// TIA Portal V19 export
FUNCTION_BLOCK "Positioning_DOL_Machine_FB"   // FB54, LAD
TITLE = OPEN LOOP POSITIONING AXIS WITH DRIVE S120 TEL.1
// stored: Access Published, MemoryReserve 100, SetENOAutomatically false
   VAR_INPUT
      AreaInterface : "AreaInterface";
      ZSI : "udt_ZoneSafetyInterface";
      DSI : "udt_DeviceSafetyInterface";
      Drive : "TAx_DriveInterface";
      DataIn : "Positioning_DOL_Machine_DataIn";
      CIn : "Positioning_DOL_Machine_CIn";
      Config : "Positioning_DOL_Machine_Config";
      HW_ID_TEL1 : HW_SUBMODULE;
   END_VAR
   VAR_OUTPUT
      MachineInterface { ExternalAccessible := 'False'; ExternalVisible := 'False'; ExternalWritable := 'False'} : "MachineInterface";
      DataOut : "Positioning_DOL_Machine_DataOut";
      COut : "Positioning_DOL_Machine_COut";
   END_VAR
   VAR_IN_OUT
      PosFeedback : "PosFbk_ITF";
      Par : "Positioning_DOL_Machine_Par";
      Pers_Data : "Positioning_DOL_Machine_Pers_Data";
      Warning : "Positioning_DOL_Machine_Wng";
      Alarm : "Positioning_DOL_Machine_Alr";
   END_VAR
   VAR
      InitDone : Bool := FALSE;
      Diag : Struct
         S120 : "TO_Diagnostic";
      END_STRUCT;
      HMI : Struct
         Sts { S7_SetPoint := 'True'} : "UDT_HMI-Sts_PosDOL-MchFB";
         B_Preset : Bool;
         B_Preset_UM2 : Bool;
         PresetPosition : LReal;
         TargetPosition : LReal;
      END_STRUCT;
      Sts : Struct
         Standstill : Bool;
         AlarmPresence : Bool;
         WarningPresence : Bool;
         Gen_Cnd : Bool;
         Minus_Cnd : Bool;
         Plus_Cnd : Bool;
         Pos_Cnd : Bool;
         Preset_Cnd : Bool;
         ActualPosition : LReal;
         Act_SysTime : DTL;
         Prv_SysTime : DTL;
      END_STRUCT;
      Ctrl : Struct
         StopDueDoorOpeningRequest : Bool;
         StopAborting : Bool;
         SafeMotionEnable : Bool;
         StopInPhase : Bool;
         StopProgrammed : Bool;
         Preset : Bool;
         Minus_Pos_Aut : Bool;
         Plus_Pos_Aut : Bool;
         Minus_Pos_Man : Bool;
         Plus_Pos_Man : Bool;
         Minus_Vel_Man : Bool;
         Plus_Vel_Man : Bool;
         MoveToPos_Aut : Bool;
         MoveToPos_Man : Bool;
         MoveToPos : Bool;
         Minus_Vel : Bool;
         Plus_Vel : Bool;
         Fan : Bool;
         Pos : LReal;
         Speed : LReal;
         SpeedPercentage : LReal;
      END_STRUCT;
      Ax : "OnOffAxis";
      S120 { S7_SetPoint := 'True'} : "SpeedMotor";
      Fan_M : "Motor";
      TON_NoPendingCmd : TON_TIME;
      TON_MinusCnd { S7_SetPoint := 'True'} : TON_TIME;
      TON_PlusCnd { S7_SetPoint := 'True'} : TON_TIME;
      TON_Fan_DelayOff : TON_TIME;
      TON_Brake_TimeOut : TON_TIME;
      S120_STW_TEL1 { ExternalAccessible := 'False'; ExternalVisible := 'False'; ExternalWritable := 'False'} : PD_TEL1_IN;
      S120_ZSW_TEL1 { ExternalAccessible := 'False'; ExternalVisible := 'False'; ExternalWritable := 'False'} : PD_TEL1_OUT;
      GETIO_STW_TEL1 { S7_SetPoint := 'True'} : GETIO;
      SETIO_ZSW_TEL1 { S7_SetPoint := 'True'} : SETIO;
      AUX : Struct
         PB_Minus : Bool;
         PB_Plus : Bool;
         PB_MoveToPos : Bool;
         B_Preset { ExternalAccessible := 'False'; ExternalVisible := 'False'; ExternalWritable := 'False'} : Bool;
         B_Preset_UM2 : Bool;
      END_STRUCT;
   END_VAR
   VAR_TEMP
      PE : Struct
         PB_Minus : Bool;
         PB_Plus : Bool;
         PB_MoveToPos : Bool;
         B_Preset : Bool;
         B_Preset_UM2 : Bool;
      END_STRUCT;
      RETVAL : Int;
      Req : Bool;
      REAL_value : Real;
   END_VAR
   VAR_TEMP   // added for the SCL form of the ladder/FBD networks
      _w1 : Bool;
      _w2 : Bool;
      _w3 : Bool;
      _w4 : Bool;
      _w5 : Bool;
   END_VAR
BEGIN

REGION Network 1 (SCL): Init
   IF NOT #InitDone THEN

       #InitDone := TRUE;

       #RETVAL := RD_SYS_T(#Sts.Act_SysTime);

       #Sts.Prv_SysTime := #Sts.Act_SysTime;

   END_IF;
END_REGION

REGION Network 2 (SCL): Reset
   IF #AreaInterface.RstAlarms THEN

       #Alarm.BrakeTimeOut := FALSE;
       #Alarm.S120_ComErr := FALSE;
       #Alarm.Ax_NotHomed := FALSE;

       #Warning.NotAutReady := FALSE;
       #Warning.MissingCnd_Minus := FALSE;
       #Warning.MissingCnd_Plus := FALSE;

   END_IF;
END_REGION

REGION Network 3 (SCL): Actual Position
   #Sts.ActualPosition := #PosFeedback.Sts.Position;
END_REGION

REGION Network 4: >
END_REGION

REGION Network 5: <<< MACHINE STOP >>>
END_REGION

REGION Network 6: Machine stop movements due door open request
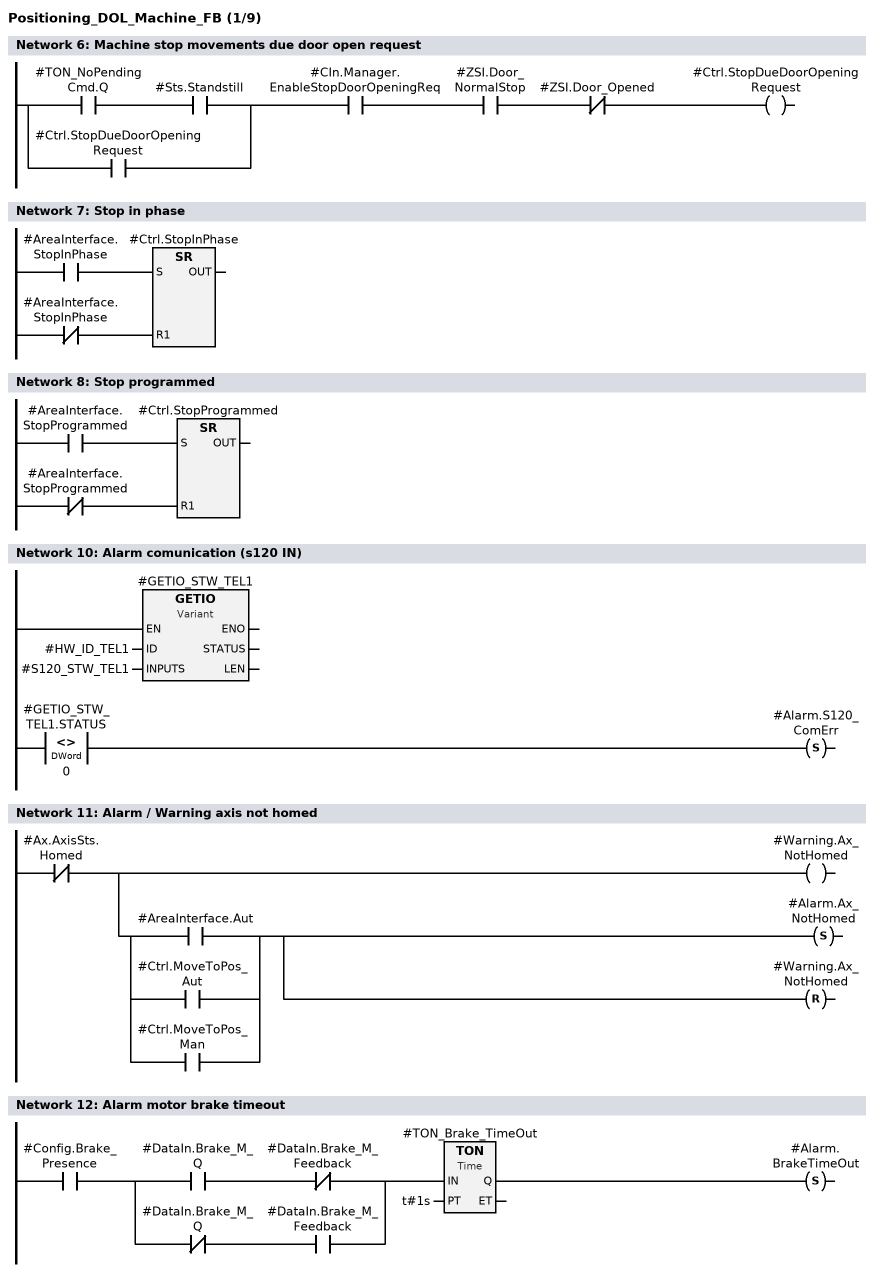
   RUNG wire#powerrail
      Contact( #TON_NoPendingCmd.Q )
      Contact( #Sts.Standstill )
      wire#w1
      Contact( #CIn.Manager.EnableStopDoorOpeningReq )
      Contact( #ZSI.Door_NormalStop )
      I_Contact( #ZSI.Door_Opened )
      Coil( #Ctrl.StopDueDoorOpeningRequest )
   END_RUNG
   RUNG wire#powerrail
      Contact( #Ctrl.StopDueDoorOpeningRequest )
   END_RUNG wire#w1
   // the same network as SCL:
   #Ctrl.StopDueDoorOpeningRequest := ((#TON_NoPendingCmd.Q AND #Sts.Standstill) OR #Ctrl.StopDueDoorOpeningRequest) AND #CIn.Manager.EnableStopDoorOpeningReq AND #ZSI.Door_NormalStop AND NOT #ZSI.Door_Opened;
END_REGION

REGION Network 7: Stop in phase
   RUNG wire#powerrail
      Contact( #AreaInterface.StopInPhase )
      S_SR(operand := #Ctrl.StopInPhase, r1 := wire#w1)
   END_RUNG
   RUNG wire#powerrail
      I_Contact( #AreaInterface.StopInPhase )
   END_RUNG wire#w1
   // the same network as SCL:
   IF #AreaInterface.StopInPhase THEN
       #Ctrl.StopInPhase := TRUE;   // SR flip-flop
   END_IF;
   IF NOT #AreaInterface.StopInPhase THEN #Ctrl.StopInPhase := FALSE; END_IF;
END_REGION

REGION Network 8: Stop programmed
   RUNG wire#powerrail
      Contact( #AreaInterface.StopProgrammed )
      S_SR(operand := #Ctrl.StopProgrammed, r1 := wire#w1)
   END_RUNG
   RUNG wire#powerrail
      I_Contact( #AreaInterface.StopProgrammed )
   END_RUNG wire#w1
   // the same network as SCL:
   IF #AreaInterface.StopProgrammed THEN
       #Ctrl.StopProgrammed := TRUE;   // SR flip-flop
   END_IF;
   IF NOT #AreaInterface.StopProgrammed THEN #Ctrl.StopProgrammed := FALSE; END_IF;
END_REGION

REGION Network 9: >
END_REGION

REGION Network 10: Alarm comunication (s120 IN)
   RUNG wire#powerrail
      { S7_Templates := "[ptr_type := Variant, id_type := HW_SUBMODULE]" } #GETIO_STW_TEL1.GETIO(ID := #HW_ID_TEL1, INPUTS := #S120_STW_TEL1, STATUS =>, LEN =>)
   END_RUNG
   RUNG wire#powerrail
      { S7_Templates := "SrcType := DWord" } NE_Contact(in1 := #GETIO_STW_TEL1.STATUS, in2 := 0)
      S_Coil( #Alarm.S120_ComErr )
   END_RUNG
   // the same network as SCL:
   #GETIO_STW_TEL1(ID := #HW_ID_TEL1, INPUTS := #S120_STW_TEL1);   // GETIO
   IF #GETIO_STW_TEL1.STATUS <> 0 THEN #Alarm.S120_ComErr := TRUE; END_IF;
END_REGION

REGION Network 11: Alarm / Warning axis not homed
   RUNG wire#powerrail
      I_Contact( #Ax.AxisSts.Homed )
      wire#w1
      Coil( #Warning.Ax_NotHomed )
   END_RUNG
   RUNG wire#w1
      Contact( #AreaInterface.Aut )
      wire#w2
      S_Coil( #Alarm.Ax_NotHomed )
   END_RUNG
   RUNG wire#w1
      Contact( #Ctrl.MoveToPos_Aut )
   END_RUNG wire#w2
   RUNG wire#w1
      Contact( #Ctrl.MoveToPos_Man )
   END_RUNG wire#w2
   RUNG wire#w2
      R_Coil( #Warning.Ax_NotHomed )
   END_RUNG
   // the same network as SCL:
   #Warning.Ax_NotHomed := NOT #Ax.AxisSts.Homed;
   IF NOT #Ax.AxisSts.Homed AND (#AreaInterface.Aut OR #Ctrl.MoveToPos_Aut OR #Ctrl.MoveToPos_Man) THEN
       #Alarm.Ax_NotHomed := TRUE;
       #Warning.Ax_NotHomed := FALSE;
   END_IF;
END_REGION

REGION Network 12: Alarm motor brake timeout
   RUNG wire#powerrail
      Contact( #Config.Brake_Presence )
      wire#w1
      Contact( #DataIn.Brake_M_Q )
      I_Contact( #DataIn.Brake_M_Feedback )
      wire#w2
      { S7_Templates := "time_type := Time" } #TON_Brake_TimeOut.TON(pt := t#1s, et =>)
      S_Coil( #Alarm.BrakeTimeOut )
   END_RUNG
   RUNG wire#w1
      I_Contact( #DataIn.Brake_M_Q )
      Contact( #DataIn.Brake_M_Feedback )
   END_RUNG wire#w2
   // the same network as SCL:
   #TON_Brake_TimeOut(IN := #Config.Brake_Presence AND ((#DataIn.Brake_M_Q AND NOT #DataIn.Brake_M_Feedback) OR (NOT #DataIn.Brake_M_Q AND #DataIn.Brake_M_Feedback)),   // TON
                      PT := t#1s);
   IF #TON_Brake_TimeOut.Q THEN #Alarm.BrakeTimeOut := TRUE; END_IF;
END_REGION

REGION Network 13: >
END_REGION

REGION Network 14: Buttons
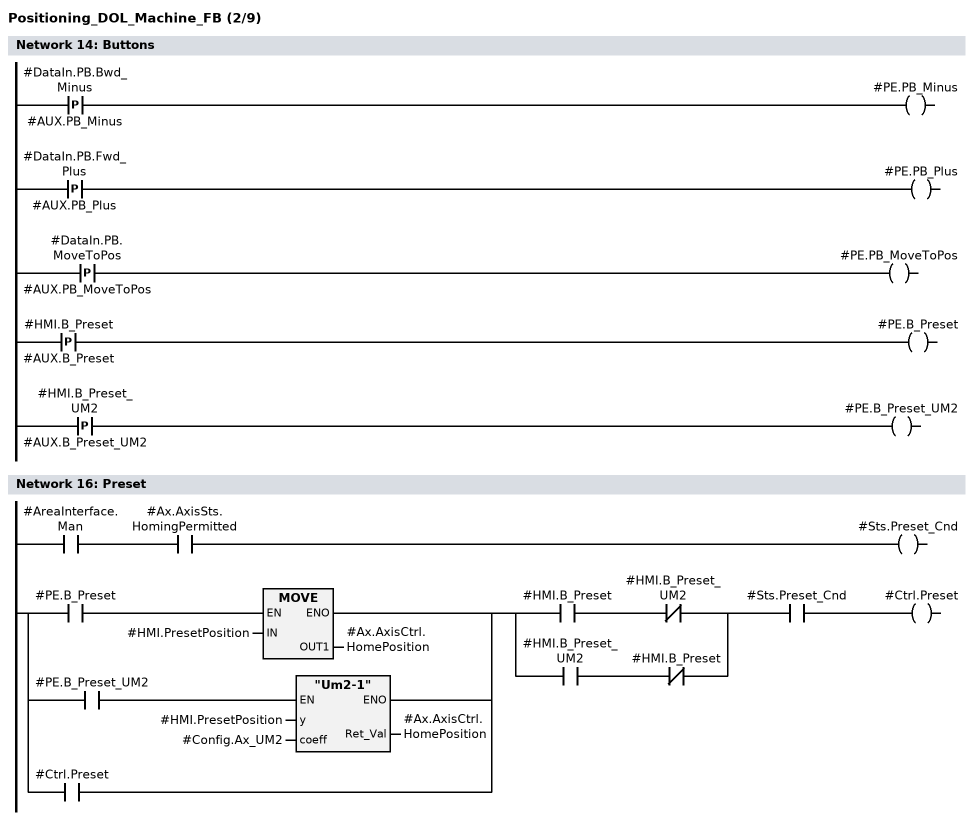
   RUNG wire#powerrail
      P_Contact(operand := #DataIn.PB.Bwd_Minus, bit := #AUX.PB_Minus)
      Coil( #PE.PB_Minus )
   END_RUNG
   RUNG wire#powerrail
      P_Contact(operand := #DataIn.PB.Fwd_Plus, bit := #AUX.PB_Plus)
      Coil( #PE.PB_Plus )
   END_RUNG
   RUNG wire#powerrail
      P_Contact(operand := #DataIn.PB.MoveToPos, bit := #AUX.PB_MoveToPos)
      Coil( #PE.PB_MoveToPos )
   END_RUNG
   RUNG wire#powerrail
      P_Contact(operand := #HMI.B_Preset, bit := #AUX.B_Preset)
      Coil( #PE.B_Preset )
   END_RUNG
   RUNG wire#powerrail
      P_Contact(operand := #HMI.B_Preset_UM2, bit := #AUX.B_Preset_UM2)
      Coil( #PE.B_Preset_UM2 )
   END_RUNG
   // the same network as SCL:
   #_w1 := #DataIn.PB.Bwd_Minus AND NOT #AUX.PB_Minus;   // rising edge of #DataIn.PB.Bwd_Minus
   #AUX.PB_Minus := #DataIn.PB.Bwd_Minus;
   #PE.PB_Minus := #_w1;
   #_w2 := #DataIn.PB.Fwd_Plus AND NOT #AUX.PB_Plus;   // rising edge of #DataIn.PB.Fwd_Plus
   #AUX.PB_Plus := #DataIn.PB.Fwd_Plus;
   #PE.PB_Plus := #_w2;
   #_w3 := #DataIn.PB.MoveToPos AND NOT #AUX.PB_MoveToPos;   // rising edge of #DataIn.PB.MoveToPos
   #AUX.PB_MoveToPos := #DataIn.PB.MoveToPos;
   #PE.PB_MoveToPos := #_w3;
   #_w4 := #HMI.B_Preset AND NOT #AUX.B_Preset;   // rising edge of #HMI.B_Preset
   #AUX.B_Preset := #HMI.B_Preset;
   #PE.B_Preset := #_w4;
   #_w5 := #HMI.B_Preset_UM2 AND NOT #AUX.B_Preset_UM2;   // rising edge of #HMI.B_Preset_UM2
   #AUX.B_Preset_UM2 := #HMI.B_Preset_UM2;
   #PE.B_Preset_UM2 := #_w5;
END_REGION

REGION Network 15: >
END_REGION

REGION Network 16: Preset
   RUNG wire#powerrail
      Contact( #AreaInterface.Man )
      Contact( #Ax.AxisSts.HomingPermitted )
      Coil( #Sts.Preset_Cnd )
   END_RUNG
   RUNG wire#powerrail
      Contact( #PE.B_Preset )
      Move(in := #HMI.PresetPosition, out1 => #Ax.AxisCtrl.HomePosition)
      wire#w1
      Contact( #HMI.B_Preset )
      I_Contact( #HMI.B_Preset_UM2 )
      wire#w2
      Contact( #Sts.Preset_Cnd )
      Coil( #Ctrl.Preset )
   END_RUNG
   RUNG wire#powerrail
      Contact( #PE.B_Preset_UM2 )
      "Um2-1"(y := #HMI.PresetPosition, coeff := #Config.Ax_UM2, Ret_Val => #Ax.AxisCtrl.HomePosition)
   END_RUNG wire#w1
   RUNG wire#powerrail
      Contact( #Ctrl.Preset )
   END_RUNG wire#w1
   RUNG wire#w1
      Contact( #HMI.B_Preset_UM2 )
      I_Contact( #HMI.B_Preset )
   END_RUNG wire#w2
   // the same network as SCL:
   #Sts.Preset_Cnd := #AreaInterface.Man AND #Ax.AxisSts.HomingPermitted;
   IF #PE.B_Preset THEN #Ax.AxisCtrl.HomePosition := #HMI.PresetPosition; END_IF;
   #Ax.AxisCtrl.HomePosition := "Um2-1"(EN := #PE.B_Preset_UM2,
                           y := #HMI.PresetPosition,
                           coeff := #Config.Ax_UM2,
                           ENO => #_w1);
   #Ctrl.Preset := (#PE.B_Preset OR #_w1 OR #Ctrl.Preset) AND ((#HMI.B_Preset AND NOT #HMI.B_Preset_UM2) OR (#HMI.B_Preset_UM2 AND NOT #HMI.B_Preset)) AND #Sts.Preset_Cnd;
END_REGION

REGION Network 17: Man
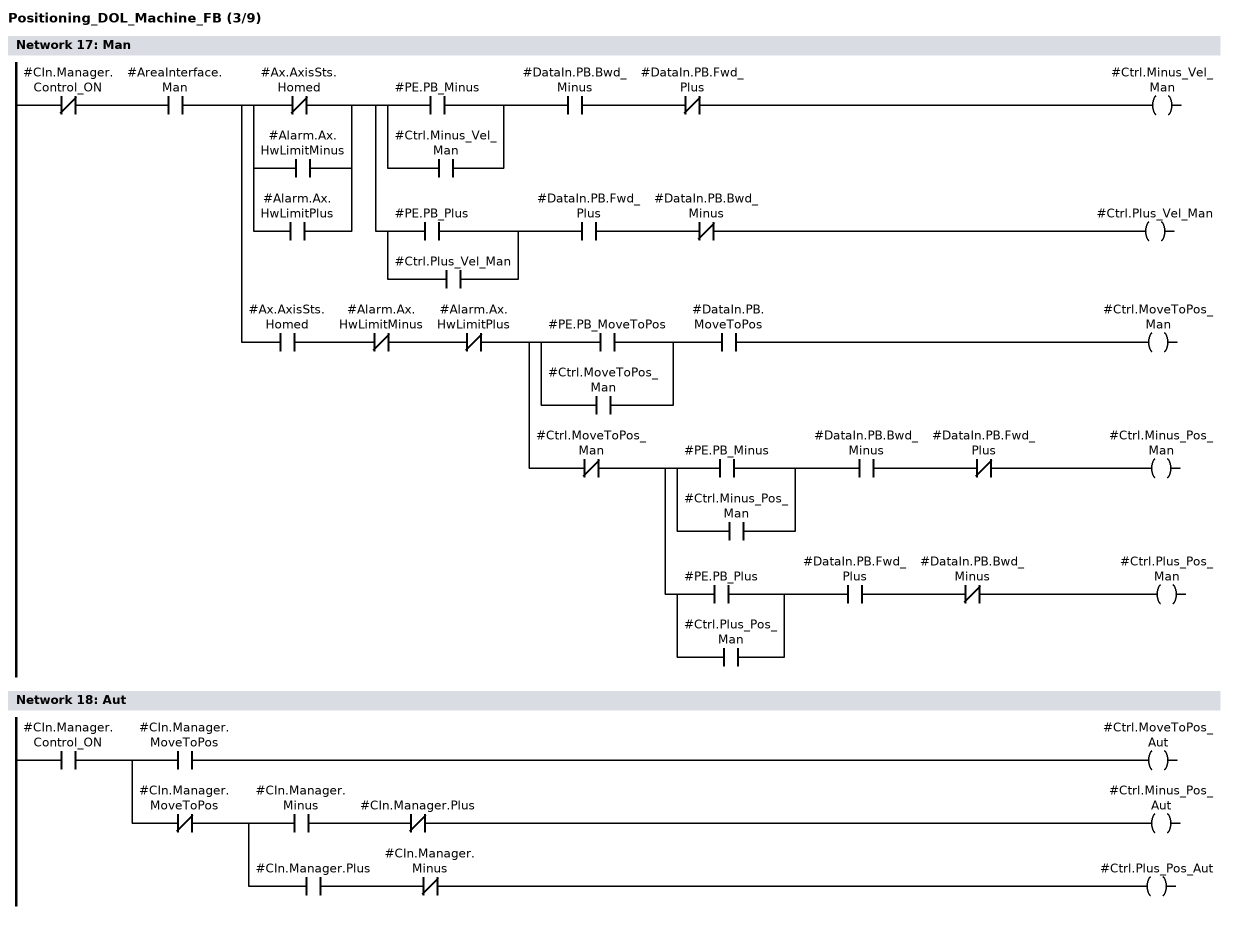
   RUNG wire#powerrail
      I_Contact( #CIn.Manager.Control_ON )
      Contact( #AreaInterface.Man )
      wire#w1
      I_Contact( #Ax.AxisSts.Homed )
      wire#w2
      Contact( #PE.PB_Minus )
      wire#w3
      Contact( #DataIn.PB.Bwd_Minus )
      I_Contact( #DataIn.PB.Fwd_Plus )
      Coil( #Ctrl.Minus_Vel_Man )
   END_RUNG
   RUNG wire#w1
      Contact( #Alarm.Ax.HwLimitMinus )
   END_RUNG wire#w2
   RUNG wire#w1
      Contact( #Alarm.Ax.HwLimitPlus )
   END_RUNG wire#w2
   RUNG wire#w2
      Contact( #Ctrl.Minus_Vel_Man )
   END_RUNG wire#w3
   RUNG wire#w2
      Contact( #PE.PB_Plus )
      wire#w4
      Contact( #DataIn.PB.Fwd_Plus )
      I_Contact( #DataIn.PB.Bwd_Minus )
      Coil( #Ctrl.Plus_Vel_Man )
   END_RUNG
   RUNG wire#w2
      Contact( #Ctrl.Plus_Vel_Man )
   END_RUNG wire#w4
   RUNG wire#w1
      Contact( #Ax.AxisSts.Homed )
      I_Contact( #Alarm.Ax.HwLimitMinus )
      I_Contact( #Alarm.Ax.HwLimitPlus )
      wire#w5
      Contact( #PE.PB_MoveToPos )
      wire#w6
      Contact( #DataIn.PB.MoveToPos )
      Coil( #Ctrl.MoveToPos_Man )
   END_RUNG
   RUNG wire#w5
      Contact( #Ctrl.MoveToPos_Man )
   END_RUNG wire#w6
   RUNG wire#w5
      I_Contact( #Ctrl.MoveToPos_Man )
      wire#w7
      Contact( #PE.PB_Minus )
      wire#w8
      Contact( #DataIn.PB.Bwd_Minus )
      I_Contact( #DataIn.PB.Fwd_Plus )
      Coil( #Ctrl.Minus_Pos_Man )
   END_RUNG
   RUNG wire#w7
      Contact( #Ctrl.Minus_Pos_Man )
   END_RUNG wire#w8
   RUNG wire#w7
      Contact( #PE.PB_Plus )
      wire#w9
      Contact( #DataIn.PB.Fwd_Plus )
      I_Contact( #DataIn.PB.Bwd_Minus )
      Coil( #Ctrl.Plus_Pos_Man )
   END_RUNG
   RUNG wire#w7
      Contact( #Ctrl.Plus_Pos_Man )
   END_RUNG wire#w9
   // the same network as SCL:
   #_w1 := NOT #CIn.Manager.Control_ON AND #AreaInterface.Man;
   #_w2 := #_w1 AND (NOT #Ax.AxisSts.Homed OR #Alarm.Ax.HwLimitMinus OR #Alarm.Ax.HwLimitPlus);
   #Ctrl.Minus_Vel_Man := #_w2 AND (#PE.PB_Minus OR #Ctrl.Minus_Vel_Man) AND #DataIn.PB.Bwd_Minus AND NOT #DataIn.PB.Fwd_Plus;
   #Ctrl.Plus_Vel_Man := #_w2 AND (#PE.PB_Plus OR #Ctrl.Plus_Vel_Man) AND #DataIn.PB.Fwd_Plus AND NOT #DataIn.PB.Bwd_Minus;
   #_w3 := #_w1 AND #Ax.AxisSts.Homed AND NOT #Alarm.Ax.HwLimitMinus AND NOT #Alarm.Ax.HwLimitPlus;
   #Ctrl.MoveToPos_Man := #_w3 AND (#PE.PB_MoveToPos OR #Ctrl.MoveToPos_Man) AND #DataIn.PB.MoveToPos;
   #_w4 := #_w3 AND NOT #Ctrl.MoveToPos_Man;
   #Ctrl.Minus_Pos_Man := #_w4 AND (#PE.PB_Minus OR #Ctrl.Minus_Pos_Man) AND #DataIn.PB.Bwd_Minus AND NOT #DataIn.PB.Fwd_Plus;
   #Ctrl.Plus_Pos_Man := #_w4 AND (#PE.PB_Plus OR #Ctrl.Plus_Pos_Man) AND #DataIn.PB.Fwd_Plus AND NOT #DataIn.PB.Bwd_Minus;
END_REGION

REGION Network 18: Aut
   RUNG wire#powerrail
      Contact( #CIn.Manager.Control_ON )
      wire#w1
      Contact( #CIn.Manager.MoveToPos )
      Coil( #Ctrl.MoveToPos_Aut )
   END_RUNG
   RUNG wire#w1
      I_Contact( #CIn.Manager.MoveToPos )
      wire#w2
      Contact( #CIn.Manager.Minus )
      I_Contact( #CIn.Manager.Plus )
      Coil( #Ctrl.Minus_Pos_Aut )
   END_RUNG
   RUNG wire#w2
      Contact( #CIn.Manager.Plus )
      I_Contact( #CIn.Manager.Minus )
      Coil( #Ctrl.Plus_Pos_Aut )
   END_RUNG
   // the same network as SCL:
   #Ctrl.MoveToPos_Aut := #CIn.Manager.Control_ON AND #CIn.Manager.MoveToPos;
   #_w1 := #CIn.Manager.Control_ON AND NOT #CIn.Manager.MoveToPos;
   #Ctrl.Minus_Pos_Aut := #_w1 AND #CIn.Manager.Minus AND NOT #CIn.Manager.Plus;
   #Ctrl.Plus_Pos_Aut := #_w1 AND #CIn.Manager.Plus AND NOT #CIn.Manager.Minus;
END_REGION

REGION Network 19: >
END_REGION

REGION Network 20 (SCL): Axis Limits
   #COut.MinPosition := #Par.Minus_Limit; //+ #Par.PosTolerance ; 

   #COut.MaxPosition := #Par.Plus_Limit; //- #Par.PosTolerance;


   IF #CIn.PositionLimits.EnableMin THEN
       #COut.MinPosition := MAX(IN1 := #COut.MinPosition, IN2 := #CIn.PositionLimits.PosMin);
   END_IF;

   IF #CIn.PositionLimits.EnableMax THEN
       #COut.MaxPosition := MIN(IN1 := #COut.MaxPosition, IN2 := #CIn.PositionLimits.PosMax);
   END_IF;
END_REGION

REGION Network 21 (SCL): Software Limit switches / External limits reached / exceed
   #COut.MinusLsSwReached := FALSE;
   #COut.PlusLsSwReached := FALSE;
   #COut.MinusLimitReached := FALSE;
   #COut.PlusLimitReached := FALSE;


   IF #Ax.AxisSts.Homed THEN

       #COut.MinusLsSwReached := #Warning.Ax.SwLimitMinus; //OR (ABS(#Sts.ActualPosition - #Par.Minus_Limit) <= #Par.PosTolerance);
       #COut.PlusLsSwReached := #Warning.Ax.SwLimitPlus; //OR (ABS(#Sts.ActualPosition - #Par.Plus_Limit) <= #Par.PosTolerance);


       IF NOT #COut.MinusLsSwReached AND #CIn.PositionLimits.EnableMin THEN

           #COut.MinusLimitReached := (#Sts.ActualPosition < #COut.MinPosition) OR (ABS(#Sts.ActualPosition - #COut.MinPosition) <= (#Par.PosTolerance/2));

       END_IF;



       IF NOT #COut.PlusLsSwReached  AND #CIn.PositionLimits.EnableMax THEN

           #COut.PlusLimitReached := (#Sts.ActualPosition > #COut.MaxPosition) OR (ABS(#Sts.ActualPosition - #COut.MaxPosition) <= (#Par.PosTolerance/2));

       END_IF;

   END_IF;
END_REGION

REGION Network 22 (SCL): Target position
   IF #CIn.Manager.Control_ON THEN


       #Ctrl.Pos := #CIn.Manager.Pos;

       IF #Ctrl.Minus_Pos_Aut THEN
           #Ctrl.Pos := #COut.MinPosition;

       ELSIF #Ctrl.Plus_Pos_Aut THEN
           #Ctrl.Pos := #COut.MaxPosition;
       END_IF;


       #HMI.TargetPosition := #Ctrl.Pos;

   ELSE


       #Ctrl.Pos := #HMI.TargetPosition;

       IF #Ctrl.Minus_Pos_Man THEN
           #Ctrl.Pos := #COut.MinPosition;
           #HMI.TargetPosition := #Ctrl.Pos;

       ELSIF #Ctrl.Plus_Pos_Man THEN
           #Ctrl.Pos := #COut.MaxPosition;
           #HMI.TargetPosition := #Ctrl.Pos;
       END_IF;

   END_IF;





   //---   



   // Dynamics limiting
   // 

   #Ctrl.Pos := LIMIT(IN := #Ctrl.Pos, MN := #COut.MinPosition, MX := #COut.MaxPosition);
END_REGION

REGION Network 23: >
END_REGION

REGION Network 24: Conditions
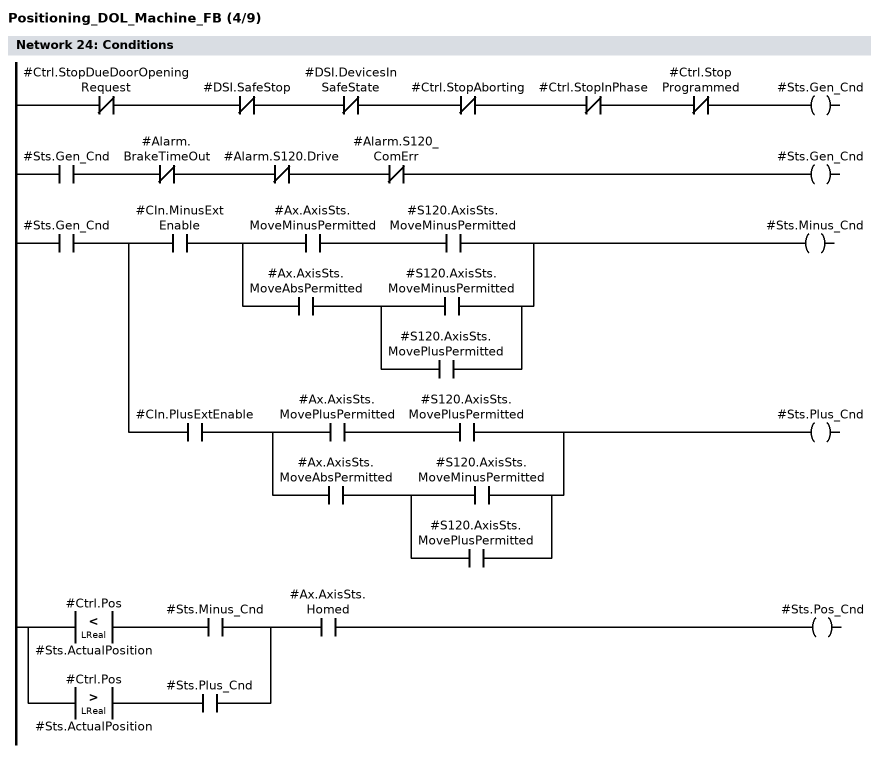
   RUNG wire#powerrail
      I_Contact( #Ctrl.StopDueDoorOpeningRequest )
      I_Contact( #DSI.SafeStop )
      I_Contact( #DSI.DevicesInSafeState )
      I_Contact( #Ctrl.StopAborting )
      I_Contact( #Ctrl.StopInPhase )
      I_Contact( #Ctrl.StopProgrammed )
      Coil( #Sts.Gen_Cnd )
   END_RUNG
   RUNG wire#powerrail
      Contact( #Sts.Gen_Cnd )
      I_Contact( #Alarm.BrakeTimeOut )
      I_Contact( #Alarm.S120.Drive )
      I_Contact( #Alarm.S120_ComErr )
      Coil( #Sts.Gen_Cnd )
   END_RUNG
   RUNG wire#powerrail
      Contact( #Sts.Gen_Cnd )
      wire#w1
      Contact( #CIn.MinusExtEnable )
      wire#w2
      Contact( #Ax.AxisSts.MoveMinusPermitted )
      Contact( #S120.AxisSts.MoveMinusPermitted )
      wire#w3
      Coil( #Sts.Minus_Cnd )
   END_RUNG
   RUNG wire#w2
      Contact( #Ax.AxisSts.MoveAbsPermitted )
      wire#w4
      Contact( #S120.AxisSts.MoveMinusPermitted )
   END_RUNG wire#w3
   RUNG wire#w4
      Contact( #S120.AxisSts.MovePlusPermitted )
   END_RUNG wire#w3
   RUNG wire#w1
      Contact( #CIn.PlusExtEnable )
      wire#w5
      Contact( #Ax.AxisSts.MovePlusPermitted )
      Contact( #S120.AxisSts.MovePlusPermitted )
      wire#w6
      Coil( #Sts.Plus_Cnd )
   END_RUNG
   RUNG wire#w5
      Contact( #Ax.AxisSts.MoveAbsPermitted )
      wire#w7
      Contact( #S120.AxisSts.MoveMinusPermitted )
   END_RUNG wire#w6
   RUNG wire#w7
      Contact( #S120.AxisSts.MovePlusPermitted )
   END_RUNG wire#w6
   RUNG wire#powerrail
      { S7_Templates := "SrcType := LReal" } LT_Contact(in1 := #Ctrl.Pos, in2 := #Sts.ActualPosition)
      Contact( #Sts.Minus_Cnd )
      wire#w8
      Contact( #Ax.AxisSts.Homed )
      Coil( #Sts.Pos_Cnd )
   END_RUNG
   RUNG wire#powerrail
      { S7_Templates := "SrcType := LReal" } GT_Contact(in1 := #Ctrl.Pos, in2 := #Sts.ActualPosition)
      Contact( #Sts.Plus_Cnd )
   END_RUNG wire#w8
   // the same network as SCL:
   #Sts.Gen_Cnd := NOT #Ctrl.StopDueDoorOpeningRequest AND NOT #DSI.SafeStop AND NOT #DSI.DevicesInSafeState AND NOT #Ctrl.StopAborting AND NOT #Ctrl.StopInPhase AND NOT #Ctrl.StopProgrammed;
   #Sts.Gen_Cnd := #Sts.Gen_Cnd AND NOT #Alarm.BrakeTimeOut AND NOT #Alarm.S120.Drive AND NOT #Alarm.S120_ComErr;
   #Sts.Minus_Cnd := #Sts.Gen_Cnd AND #CIn.MinusExtEnable AND ((#Ax.AxisSts.MoveMinusPermitted AND #S120.AxisSts.MoveMinusPermitted) OR (#Ax.AxisSts.MoveAbsPermitted AND (#S120.AxisSts.MoveMinusPermitted OR #S120.AxisSts.MovePlusPermitted)));
   #Sts.Plus_Cnd := #Sts.Gen_Cnd AND #CIn.PlusExtEnable AND ((#Ax.AxisSts.MovePlusPermitted AND #S120.AxisSts.MovePlusPermitted) OR (#Ax.AxisSts.MoveAbsPermitted AND (#S120.AxisSts.MoveMinusPermitted OR #S120.AxisSts.MovePlusPermitted)));
   #Sts.Pos_Cnd := (((#Ctrl.Pos < #Sts.ActualPosition) AND #Sts.Minus_Cnd) OR ((#Ctrl.Pos > #Sts.ActualPosition) AND #Sts.Plus_Cnd)) AND #Ax.AxisSts.Homed;
END_REGION

REGION Network 25: >
END_REGION

REGION Network 26: <<< ON/OFF AXIS >>>
END_REGION

REGION Network 27: On/Off Axis - Controls
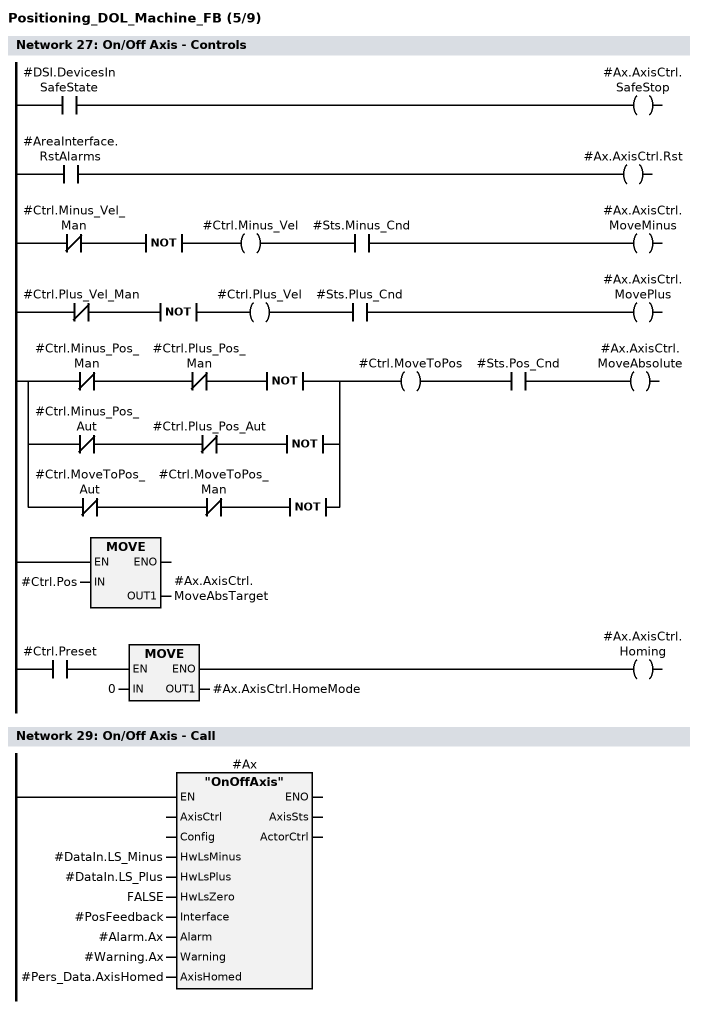
   RUNG wire#powerrail
      Contact( #DSI.DevicesInSafeState )
      Coil( #Ax.AxisCtrl.SafeStop )
   END_RUNG
   RUNG wire#powerrail
      Contact( #AreaInterface.RstAlarms )
      Coil( #Ax.AxisCtrl.Rst )
   END_RUNG
   RUNG wire#powerrail
      I_Contact( #Ctrl.Minus_Vel_Man )
      Not()
      Coil( #Ctrl.Minus_Vel )
      Contact( #Sts.Minus_Cnd )
      Coil( #Ax.AxisCtrl.MoveMinus )
   END_RUNG
   RUNG wire#powerrail
      I_Contact( #Ctrl.Plus_Vel_Man )
      Not()
      Coil( #Ctrl.Plus_Vel )
      Contact( #Sts.Plus_Cnd )
      Coil( #Ax.AxisCtrl.MovePlus )
   END_RUNG
   RUNG wire#powerrail
      I_Contact( #Ctrl.Minus_Pos_Man )
      I_Contact( #Ctrl.Plus_Pos_Man )
      Not()
      wire#w1
      Coil( #Ctrl.MoveToPos )
      Contact( #Sts.Pos_Cnd )
      Coil( #Ax.AxisCtrl.MoveAbsolute )
   END_RUNG
   RUNG wire#powerrail
      I_Contact( #Ctrl.Minus_Pos_Aut )
      I_Contact( #Ctrl.Plus_Pos_Aut )
      Not()
   END_RUNG wire#w1
   RUNG wire#powerrail
      I_Contact( #Ctrl.MoveToPos_Aut )
      I_Contact( #Ctrl.MoveToPos_Man )
      Not()
   END_RUNG wire#w1
   RUNG wire#powerrail
      Move(in := #Ctrl.Pos, out1 => #Ax.AxisCtrl.MoveAbsTarget)
   END_RUNG
   RUNG wire#powerrail
      Contact( #Ctrl.Preset )
      Move(in := 0, out1 => #Ax.AxisCtrl.HomeMode)
      Coil( #Ax.AxisCtrl.Homing )
   END_RUNG
   // the same network as SCL:
   #Ax.AxisCtrl.SafeStop := #DSI.DevicesInSafeState;
   #Ax.AxisCtrl.Rst := #AreaInterface.RstAlarms;
   #Ctrl.Minus_Vel := NOT (NOT #Ctrl.Minus_Vel_Man);
   #Ax.AxisCtrl.MoveMinus := NOT (NOT #Ctrl.Minus_Vel_Man) AND #Sts.Minus_Cnd;
   #Ctrl.Plus_Vel := NOT (NOT #Ctrl.Plus_Vel_Man);
   #Ax.AxisCtrl.MovePlus := NOT (NOT #Ctrl.Plus_Vel_Man) AND #Sts.Plus_Cnd;
   #Ctrl.MoveToPos := NOT (NOT #Ctrl.Minus_Pos_Man AND NOT #Ctrl.Plus_Pos_Man) OR NOT (NOT #Ctrl.Minus_Pos_Aut AND NOT #Ctrl.Plus_Pos_Aut) OR NOT (NOT #Ctrl.MoveToPos_Aut AND NOT #Ctrl.MoveToPos_Man);
   #Ax.AxisCtrl.MoveAbsolute := #Ctrl.MoveToPos AND #Sts.Pos_Cnd;
   #Ax.AxisCtrl.MoveAbsTarget := #Ctrl.Pos;
   IF #Ctrl.Preset THEN #Ax.AxisCtrl.HomeMode := 0; END_IF;
   #Ax.AxisCtrl.Homing := #Ctrl.Preset;
END_REGION

REGION Network 28 (SCL): On/Off Axis - Configuration
   #Ax.Config := #Config.Ax;

   #Ax.Config.limitMinus := #Par.Minus_Limit;
   #Ax.Config.limitPlus := #Par.Plus_Limit;

   #Ax.Config.ToleranceWindow := #Par.PosTolerance;
   #Ax.Config.PreCutOff := #Par.PreCutOff;
   #Ax.Config.PreEndMedSpeed := #Par.PreEndMedSpeed;
   #Ax.Config.PreEndLowSpeed := #Par.PreEndLowSpeed;


   #Ax.Config.StandStillDelay := DINT_TO_TIME(LREAL_TO_DINT(#Config.S120.DecTime + 0.1));



   IF #Config.CyclicOBTime_ms <= 0.0 THEN

       #Sts.Prv_SysTime := #Sts.Act_SysTime;

       #RETVAL := RD_SYS_T(#Sts.Act_SysTime);

       #Ax.Config.RecallTime := UDINT_TO_LREAL(TIME_TO_UDINT(T_DIFF(IN1 := #Sts.Act_SysTime, IN2 := #Sts.Prv_SysTime)));
       IF #Ax.Config.RecallTime <= 1 THEN
           #Ax.Config.RecallTime := 1;
       END_IF;
   ELSE

       #Ax.Config.RecallTime := #Config.CyclicOBTime_ms;

   END_IF;
END_REGION

REGION Network 29: On/Off Axis - Call
   RUNG wire#powerrail
      #Ax(AxisCtrl :=, Config :=, HwLsMinus := #DataIn.LS_Minus, HwLsPlus := #DataIn.LS_Plus, HwLsZero := FALSE, Interface := #PosFeedback, Alarm := #Alarm.Ax, Warning := #Warning.Ax, AxisHomed := #Pers_Data.AxisHomed, AxisSts =>, ActorCtrl =>)
   END_RUNG
   // the same network as SCL:
   #Ax(HwLsMinus := #DataIn.LS_Minus,   // "OnOffAxis"
       HwLsPlus := #DataIn.LS_Plus,
       HwLsZero := FALSE,
       Interface := #PosFeedback,
       Alarm := #Alarm.Ax,
       Warning := #Warning.Ax,
       AxisHomed := #Pers_Data.AxisHomed);
END_REGION

REGION Network 30 (SCL): On/Off Axis -Reset Wanrning

   #Warning.Ax.SwLimitMinus := (ABS(#Sts.ActualPosition - #Par.Minus_Limit) <= (#Par.PosTolerance / 2));
   #Warning.Ax.SwLimitPlus := (ABS(#Sts.ActualPosition - #Par.Plus_Limit) <= (#Par.PosTolerance / 2));
END_REGION

REGION Network 31 (SCL): S120 - Velocity & Dynamics
   #Ctrl.SpeedPercentage := #Par.Man_Speed;

   IF #CIn.Manager.Control_ON THEN
       #Ctrl.SpeedPercentage := #CIn.Manager.Speed;
   END_IF;

   #Ctrl.SpeedPercentage := MIN(IN1 := #Ctrl.SpeedPercentage, IN2 := 100.0);
   #Ctrl.SpeedPercentage := MAX(IN1 := #Ctrl.SpeedPercentage, IN2 := 0.0);


   #Ctrl.Speed := 0.0;


   IF #Ax.ActorCtrl.CmdLowSpeed THEN

       #Ctrl.Speed := (#Par.LowSpeed / 100.0) * #Config.S120.SpeedMotor.ReferenceVelocity;


       IF NOT #Ax.AxisCtrl.MoveAbsolute THEN

           #Ctrl.Speed := #Ctrl.Speed * #Ctrl.SpeedPercentage / 100.0;
       END_IF;


   ELSIF #Ax.ActorCtrl.CmdMediumSpeed THEN

       #Ctrl.Speed := (#Par.MedSpeed / 100.0) * #Config.S120.SpeedMotor.ReferenceVelocity;

       #Ctrl.Speed := #Ctrl.Speed * #Ctrl.SpeedPercentage / 100.0;


   ELSIF #Ax.ActorCtrl.CmdHighSpeed THEN

       #Ctrl.Speed := (#Par.HighSpeed / 100.0) * #Config.S120.SpeedMotor.ReferenceVelocity;

       #Ctrl.Speed := #Ctrl.Speed * #Ctrl.SpeedPercentage / 100.0;
   END_IF;



   // Brake not open... Velocity  = 0.0
   // 
   IF #Config.Brake_Presence AND NOT #DataIn.Brake_M_Feedback THEN
       #Ctrl.Speed := 0.0;
   END_IF;



   #S120.AxisCtrl.Velocity := MIN(IN1 := #Ctrl.Speed , IN2 := #Config.S120.SpeedMotor.ReferenceVelocity);

   #S120.AxisCtrl.Acceleration := #Config.S120.SpeedMotor.ReferenceVelocity / 60.0 / #Config.S120.AccTime;
   #S120.AxisCtrl.Deceleration := #Config.S120.SpeedMotor.ReferenceVelocity / 60.0 / #Config.S120.DecTime;
END_REGION

REGION Network 32: S120 - Control
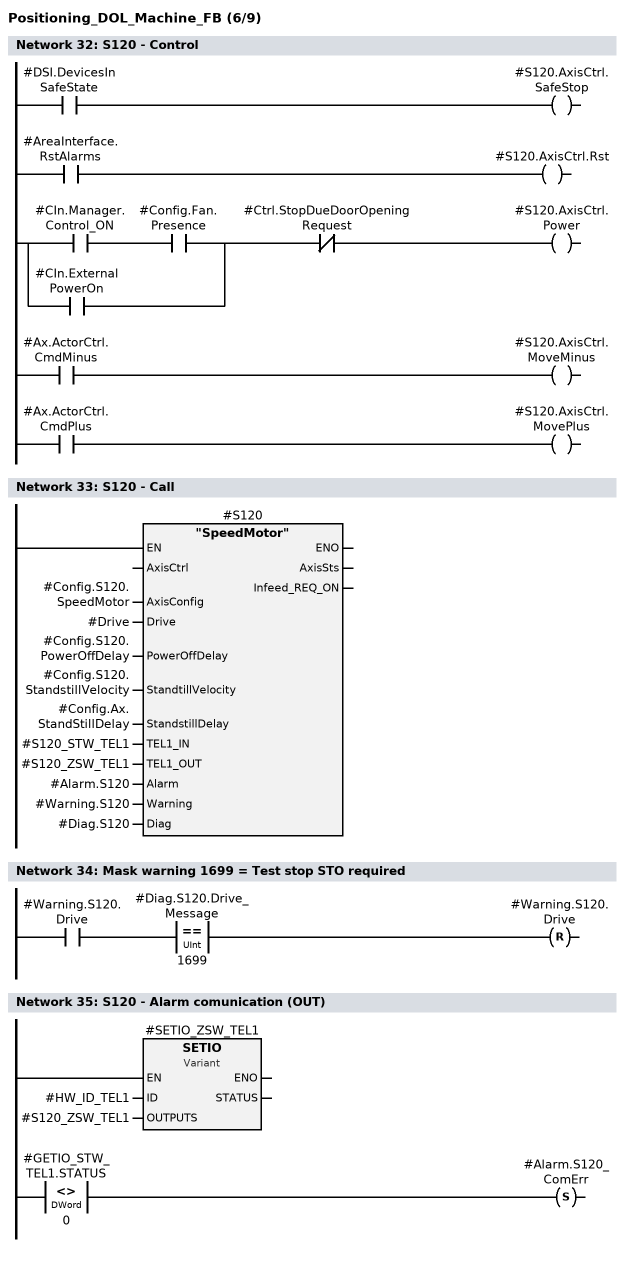
   RUNG wire#powerrail
      Contact( #DSI.DevicesInSafeState )
      Coil( #S120.AxisCtrl.SafeStop )
   END_RUNG
   RUNG wire#powerrail
      Contact( #AreaInterface.RstAlarms )
      Coil( #S120.AxisCtrl.Rst )
   END_RUNG
   RUNG wire#powerrail
      Contact( #CIn.Manager.Control_ON )
      Contact( #Config.Fan.Presence )
      wire#w1
      I_Contact( #Ctrl.StopDueDoorOpeningRequest )
      Coil( #S120.AxisCtrl.Power )
   END_RUNG
   RUNG wire#powerrail
      Contact( #CIn.ExternalPowerOn )
   END_RUNG wire#w1
   RUNG wire#powerrail
      Contact( #Ax.ActorCtrl.CmdMinus )
      Coil( #S120.AxisCtrl.MoveMinus )
   END_RUNG
   RUNG wire#powerrail
      Contact( #Ax.ActorCtrl.CmdPlus )
      Coil( #S120.AxisCtrl.MovePlus )
   END_RUNG
   // the same network as SCL:
   #S120.AxisCtrl.SafeStop := #DSI.DevicesInSafeState;
   #S120.AxisCtrl.Rst := #AreaInterface.RstAlarms;
   #S120.AxisCtrl.Power := ((#CIn.Manager.Control_ON AND #Config.Fan.Presence) OR #CIn.ExternalPowerOn) AND NOT #Ctrl.StopDueDoorOpeningRequest;
   #S120.AxisCtrl.MoveMinus := #Ax.ActorCtrl.CmdMinus;
   #S120.AxisCtrl.MovePlus := #Ax.ActorCtrl.CmdPlus;
END_REGION

REGION Network 33: S120 - Call
   RUNG wire#powerrail
      #S120(AxisCtrl :=, AxisConfig := #Config.S120.SpeedMotor, Drive := #Drive, PowerOffDelay := #Config.S120.PowerOffDelay, StandtillVelocity := #Config.S120.StandstillVelocity, StandstillDelay := #Config.Ax.StandStillDelay, TEL1_IN := #S120_STW_TEL1, TEL1_OUT := #S120_ZSW_TEL1, Alarm := #Alarm.S120, Warning := #Warning.S120, Diag := #Diag.S120, AxisSts =>, Infeed_REQ_ON =>)
   END_RUNG
   // the same network as SCL:
   #S120(AxisConfig := #Config.S120.SpeedMotor,   // "SpeedMotor"
         Drive := #Drive,
         PowerOffDelay := #Config.S120.PowerOffDelay,
         StandtillVelocity := #Config.S120.StandstillVelocity,
         StandstillDelay := #Config.Ax.StandStillDelay,
         TEL1_IN := #S120_STW_TEL1,
         TEL1_OUT := #S120_ZSW_TEL1,
         Alarm := #Alarm.S120,
         Warning := #Warning.S120,
         Diag := #Diag.S120);
END_REGION

REGION Network 34: Mask warning 1699 = Test stop STO required
   RUNG wire#powerrail
      Contact( #Warning.S120.Drive )
      { S7_Templates := "SrcType := UInt" } EQ_Contact(in1 := #Diag.S120.Drive_Message, in2 := 1699)
      R_Coil( #Warning.S120.Drive )
   END_RUNG
   // the same network as SCL:
   IF #Warning.S120.Drive AND (#Diag.S120.Drive_Message = 1699) THEN #Warning.S120.Drive := FALSE; END_IF;
END_REGION

REGION Network 35: S120 - Alarm comunication (OUT)
   RUNG wire#powerrail
      { S7_Templates := "[card := 0, ptr_type := Variant, id_type := HW_SUBMODULE]" } #SETIO_ZSW_TEL1.SETIO(ID := #HW_ID_TEL1, OUTPUTS := #S120_ZSW_TEL1, STATUS =>)
   END_RUNG
   RUNG wire#powerrail
      { S7_Templates := "SrcType := DWord" } NE_Contact(in1 := #GETIO_STW_TEL1.STATUS, in2 := 0)
      S_Coil( #Alarm.S120_ComErr )
   END_RUNG
   // the same network as SCL:
   #SETIO_ZSW_TEL1(ID := #HW_ID_TEL1, OUTPUTS := #S120_ZSW_TEL1);   // SETIO
   IF #GETIO_STW_TEL1.STATUS <> 0 THEN #Alarm.S120_ComErr := TRUE; END_IF;
END_REGION

REGION Network 36: <<< MOTOR FAN >>>
END_REGION

REGION Network 37: Run
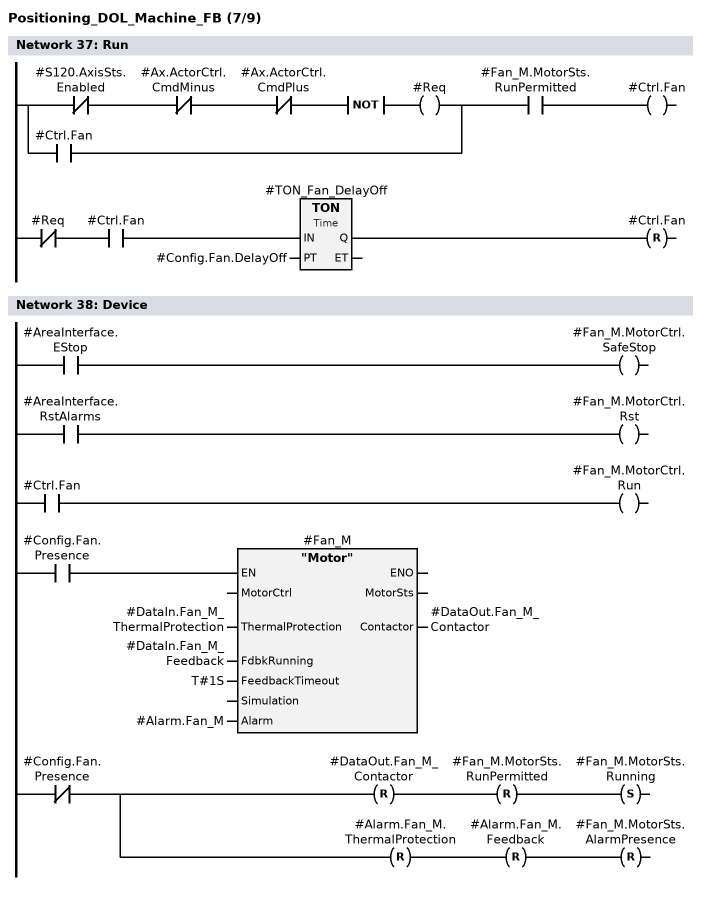
   RUNG wire#powerrail
      I_Contact( #S120.AxisSts.Enabled )
      I_Contact( #Ax.ActorCtrl.CmdMinus )
      I_Contact( #Ax.ActorCtrl.CmdPlus )
      Not()
      Coil( #Req )
      wire#w1
      Contact( #Fan_M.MotorSts.RunPermitted )
      Coil( #Ctrl.Fan )
   END_RUNG
   RUNG wire#powerrail
      Contact( #Ctrl.Fan )
   END_RUNG wire#w1
   RUNG wire#powerrail
      I_Contact( #Req )
      Contact( #Ctrl.Fan )
      { S7_Templates := "time_type := Time" } #TON_Fan_DelayOff.TON(pt := #Config.Fan.DelayOff, et =>)
      R_Coil( #Ctrl.Fan )
   END_RUNG
   // the same network as SCL:
   #Req := NOT (NOT #S120.AxisSts.Enabled AND NOT #Ax.ActorCtrl.CmdMinus AND NOT #Ax.ActorCtrl.CmdPlus);
   #Ctrl.Fan := (#Req OR #Ctrl.Fan) AND #Fan_M.MotorSts.RunPermitted;
   #TON_Fan_DelayOff(IN := NOT #Req AND #Ctrl.Fan, PT := #Config.Fan.DelayOff);   // TON
   IF #TON_Fan_DelayOff.Q THEN #Ctrl.Fan := FALSE; END_IF;
END_REGION

REGION Network 38: Device
   RUNG wire#powerrail
      Contact( #AreaInterface.EStop )
      Coil( #Fan_M.MotorCtrl.SafeStop )
   END_RUNG
   RUNG wire#powerrail
      Contact( #AreaInterface.RstAlarms )
      Coil( #Fan_M.MotorCtrl.Rst )
   END_RUNG
   RUNG wire#powerrail
      Contact( #Ctrl.Fan )
      Coil( #Fan_M.MotorCtrl.Run )
   END_RUNG
   RUNG wire#powerrail
      Contact( #Config.Fan.Presence )
      #Fan_M(MotorCtrl :=, ThermalProtection := #DataIn.Fan_M_ThermalProtection, FdbkRunning := #DataIn.Fan_M_Feedback, FeedbackTimeout := T#1S, Simulation :=, Alarm := #Alarm.Fan_M, MotorSts =>, Contactor => #DataOut.Fan_M_Contactor)
   END_RUNG
   RUNG wire#powerrail
      I_Contact( #Config.Fan.Presence )
      wire#w1
      R_Coil( #DataOut.Fan_M_Contactor )
      R_Coil( #Fan_M.MotorSts.RunPermitted )
      S_Coil( #Fan_M.MotorSts.Running )
   END_RUNG
   RUNG wire#w1
      R_Coil( #Alarm.Fan_M.ThermalProtection )
      R_Coil( #Alarm.Fan_M.Feedback )
      R_Coil( #Fan_M.MotorSts.AlarmPresence )
   END_RUNG
   // the same network as SCL:
   #Fan_M.MotorCtrl.SafeStop := #AreaInterface.EStop;
   #Fan_M.MotorCtrl.Rst := #AreaInterface.RstAlarms;
   #Fan_M.MotorCtrl.Run := #Ctrl.Fan;
   IF #Config.Fan.Presence THEN
       #Fan_M(ThermalProtection := #DataIn.Fan_M_ThermalProtection,   // "Motor"
              FdbkRunning := #DataIn.Fan_M_Feedback,
              FeedbackTimeout := T#1S,
              Alarm := #Alarm.Fan_M,
              Contactor => #DataOut.Fan_M_Contactor);
   END_IF;
   IF NOT #Config.Fan.Presence THEN
       #DataOut.Fan_M_Contactor := FALSE;
       #Fan_M.MotorSts.RunPermitted := FALSE;
       #Fan_M.MotorSts.Running := TRUE;
       #Alarm.Fan_M.ThermalProtection := FALSE;
       #Alarm.Fan_M.Feedback := FALSE;
       #Fan_M.MotorSts.AlarmPresence := FALSE;
   END_IF;
END_REGION

REGION Network 39: >
END_REGION

REGION Network 40: >
END_REGION

REGION Network 41: Coordination Out
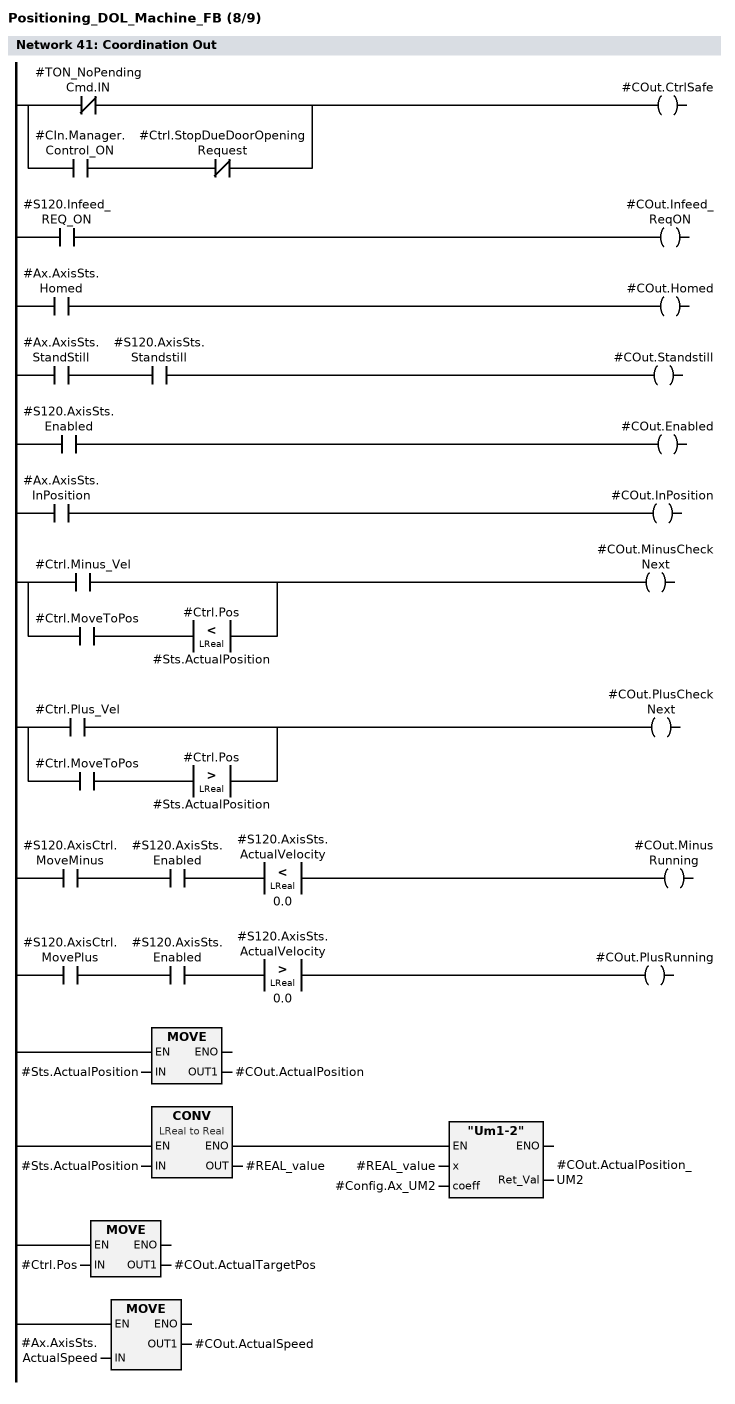
   RUNG wire#powerrail
      I_Contact( #TON_NoPendingCmd.IN )
      wire#w1
      Coil( #COut.CtrlSafe )
   END_RUNG
   RUNG wire#powerrail
      Contact( #CIn.Manager.Control_ON )
      I_Contact( #Ctrl.StopDueDoorOpeningRequest )
   END_RUNG wire#w1
   RUNG wire#powerrail
      Contact( #S120.Infeed_REQ_ON )
      Coil( #COut.Infeed_ReqON )
   END_RUNG
   RUNG wire#powerrail
      Contact( #Ax.AxisSts.Homed )
      Coil( #COut.Homed )
   END_RUNG
   RUNG wire#powerrail
      Contact( #Ax.AxisSts.StandStill )
      Contact( #S120.AxisSts.Standstill )
      Coil( #COut.Standstill )
   END_RUNG
   RUNG wire#powerrail
      Contact( #S120.AxisSts.Enabled )
      Coil( #COut.Enabled )
   END_RUNG
   RUNG wire#powerrail
      Contact( #Ax.AxisSts.InPosition )
      Coil( #COut.InPosition )
   END_RUNG
   RUNG wire#powerrail
      Contact( #Ctrl.Minus_Vel )
      wire#w2
      Coil( #COut.MinusCheckNext )
   END_RUNG
   RUNG wire#powerrail
      Contact( #Ctrl.MoveToPos )
      { S7_Templates := "SrcType := LReal" } LT_Contact(in1 := #Ctrl.Pos, in2 := #Sts.ActualPosition)
   END_RUNG wire#w2
   RUNG wire#powerrail
      Contact( #Ctrl.Plus_Vel )
      wire#w3
      Coil( #COut.PlusCheckNext )
   END_RUNG
   RUNG wire#powerrail
      Contact( #Ctrl.MoveToPos )
      { S7_Templates := "SrcType := LReal" } GT_Contact(in1 := #Ctrl.Pos, in2 := #Sts.ActualPosition)
   END_RUNG wire#w3
   RUNG wire#powerrail
      Contact( #S120.AxisCtrl.MoveMinus )
      Contact( #S120.AxisSts.Enabled )
      { S7_Templates := "SrcType := LReal" } LT_Contact(in1 := #S120.AxisSts.ActualVelocity, in2 := 0.0)
      Coil( #COut.MinusRunning )
   END_RUNG
   RUNG wire#powerrail
      Contact( #S120.AxisCtrl.MovePlus )
      Contact( #S120.AxisSts.Enabled )
      { S7_Templates := "SrcType := LReal" } GT_Contact(in1 := #S120.AxisSts.ActualVelocity, in2 := 0.0)
      Coil( #COut.PlusRunning )
   END_RUNG
   RUNG wire#powerrail
      Move(in := #Sts.ActualPosition, out1 => #COut.ActualPosition)
   END_RUNG
   RUNG wire#powerrail
      { S7_Templates := "[SrcType := LReal, DestType := Real]" } Convert(in := #Sts.ActualPosition, out => #REAL_value)
      "Um1-2"(x := #REAL_value, coeff := #Config.Ax_UM2, Ret_Val => #COut.ActualPosition_UM2)
   END_RUNG
   RUNG wire#powerrail
      Move(in := #Ctrl.Pos, out1 => #COut.ActualTargetPos)
   END_RUNG
   RUNG wire#powerrail
      Move(in := #Ax.AxisSts.ActualSpeed, out1 => #COut.ActualSpeed)
   END_RUNG
   // the same network as SCL:
   #COut.CtrlSafe := NOT #TON_NoPendingCmd.IN OR (#CIn.Manager.Control_ON AND NOT #Ctrl.StopDueDoorOpeningRequest);
   #COut.Infeed_ReqON := #S120.Infeed_REQ_ON;
   #COut.Homed := #Ax.AxisSts.Homed;
   #COut.Standstill := #Ax.AxisSts.StandStill AND #S120.AxisSts.Standstill;
   #COut.Enabled := #S120.AxisSts.Enabled;
   #COut.InPosition := #Ax.AxisSts.InPosition;
   #COut.MinusCheckNext := #Ctrl.Minus_Vel OR (#Ctrl.MoveToPos AND (#Ctrl.Pos < #Sts.ActualPosition));
   #COut.PlusCheckNext := #Ctrl.Plus_Vel OR (#Ctrl.MoveToPos AND (#Ctrl.Pos > #Sts.ActualPosition));
   #COut.MinusRunning := #S120.AxisCtrl.MoveMinus AND #S120.AxisSts.Enabled AND (#S120.AxisSts.ActualVelocity < 0.0);
   #COut.PlusRunning := #S120.AxisCtrl.MovePlus AND #S120.AxisSts.Enabled AND (#S120.AxisSts.ActualVelocity > 0.0);
   #COut.ActualPosition := #Sts.ActualPosition;
   #REAL_value := LREAL_TO_REAL(#Sts.ActualPosition);
   #COut.ActualPosition_UM2 := "Um1-2"(x := #REAL_value, coeff := #Config.Ax_UM2);
   #COut.ActualTargetPos := #Ctrl.Pos;
   #COut.ActualSpeed := #Ax.AxisSts.ActualSpeed;
END_REGION

REGION Network 42 (SCL): Coordination Out - Actual speed drive 0-100 %
   #COut.ActualSpeed_Drive := #S120.AxisSts.ActualVelocity / #Config.S120.SpeedMotor.ReferenceVelocity * 100.0;
END_REGION

REGION Network 43: Warning Missing conditions
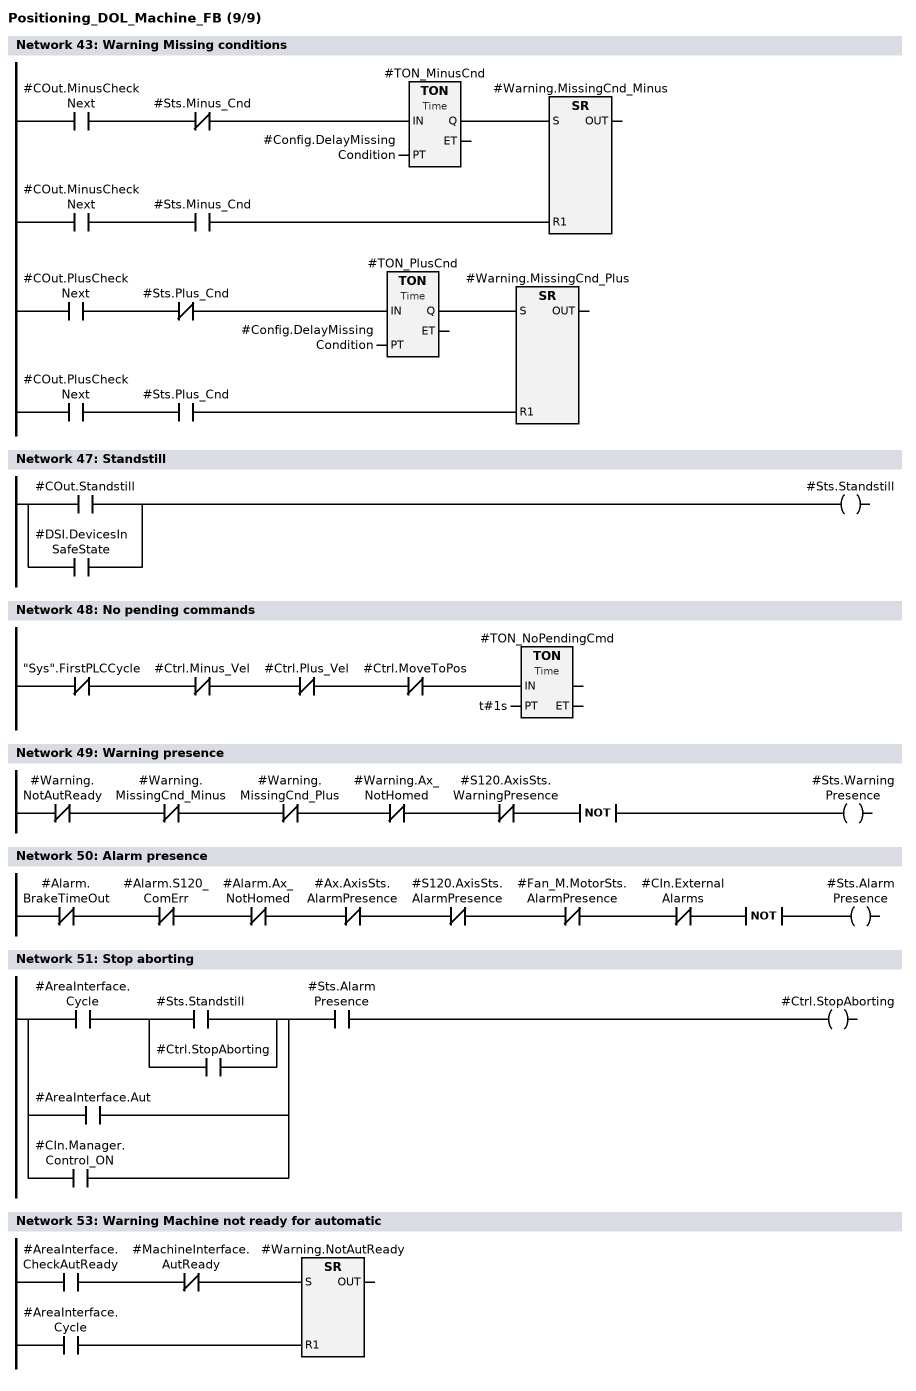
   RUNG wire#powerrail
      Contact( #COut.MinusCheckNext )
      I_Contact( #Sts.Minus_Cnd )
      { S7_Templates := "time_type := Time" } #TON_MinusCnd.TON(pt := #Config.DelayMissingCondition, et =>)
      S_SR(operand := #Warning.MissingCnd_Minus, r1 := wire#w1)
   END_RUNG
   RUNG wire#powerrail
      Contact( #COut.MinusCheckNext )
      Contact( #Sts.Minus_Cnd )
   END_RUNG wire#w1
   RUNG wire#powerrail
      Contact( #COut.PlusCheckNext )
      I_Contact( #Sts.Plus_Cnd )
      { S7_Templates := "time_type := Time" } #TON_PlusCnd.TON(pt := #Config.DelayMissingCondition, et =>)
      S_SR(operand := #Warning.MissingCnd_Plus, r1 := wire#w2)
   END_RUNG
   RUNG wire#powerrail
      Contact( #COut.PlusCheckNext )
      Contact( #Sts.Plus_Cnd )
   END_RUNG wire#w2
   // the same network as SCL:
   #TON_MinusCnd(IN := #COut.MinusCheckNext AND NOT #Sts.Minus_Cnd, PT := #Config.DelayMissingCondition);   // TON
   IF #TON_MinusCnd.Q THEN
       #Warning.MissingCnd_Minus := TRUE;   // SR flip-flop
   END_IF;
   IF #COut.MinusCheckNext AND #Sts.Minus_Cnd THEN #Warning.MissingCnd_Minus := FALSE; END_IF;
   #TON_PlusCnd(IN := #COut.PlusCheckNext AND NOT #Sts.Plus_Cnd, PT := #Config.DelayMissingCondition);   // TON
   IF #TON_PlusCnd.Q THEN
       #Warning.MissingCnd_Plus := TRUE;   // SR flip-flop
   END_IF;
   IF #COut.PlusCheckNext AND #Sts.Plus_Cnd THEN #Warning.MissingCnd_Plus := FALSE; END_IF;
END_REGION

REGION Network 44: >
END_REGION

REGION Network 45: >
END_REGION

REGION Network 46: <<< MACHINE STATUS >>>
END_REGION

REGION Network 47: Standstill
   RUNG wire#powerrail
      Contact( #COut.Standstill )
      wire#w1
      Coil( #Sts.Standstill )
   END_RUNG
   RUNG wire#powerrail
      Contact( #DSI.DevicesInSafeState )
   END_RUNG wire#w1
   // the same network as SCL:
   #Sts.Standstill := #COut.Standstill OR #DSI.DevicesInSafeState;
END_REGION

REGION Network 48: No pending commands
   RUNG wire#powerrail
      I_Contact( "Sys".FirstPLCCycle )
      I_Contact( #Ctrl.Minus_Vel )
      I_Contact( #Ctrl.Plus_Vel )
      I_Contact( #Ctrl.MoveToPos )
      { S7_Templates := "time_type := Time" } #TON_NoPendingCmd.TON(pt := t#1s, et =>)
   END_RUNG
   // the same network as SCL:
   #TON_NoPendingCmd(IN := NOT "Sys".FirstPLCCycle AND NOT #Ctrl.Minus_Vel AND NOT #Ctrl.Plus_Vel AND NOT #Ctrl.MoveToPos,   // TON
                     PT := t#1s);
END_REGION

REGION Network 49: Warning presence
   RUNG wire#powerrail
      I_Contact( #Warning.NotAutReady )
      I_Contact( #Warning.MissingCnd_Minus )
      I_Contact( #Warning.MissingCnd_Plus )
      I_Contact( #Warning.Ax_NotHomed )
      I_Contact( #S120.AxisSts.WarningPresence )
      Not()
      Coil( #Sts.WarningPresence )
   END_RUNG
   // the same network as SCL:
   #Sts.WarningPresence := NOT (NOT #Warning.NotAutReady AND NOT #Warning.MissingCnd_Minus AND NOT #Warning.MissingCnd_Plus AND NOT #Warning.Ax_NotHomed AND NOT #S120.AxisSts.WarningPresence);
END_REGION

REGION Network 50: Alarm presence
   RUNG wire#powerrail
      I_Contact( #Alarm.BrakeTimeOut )
      I_Contact( #Alarm.S120_ComErr )
      I_Contact( #Alarm.Ax_NotHomed )
      I_Contact( #Ax.AxisSts.AlarmPresence )
      I_Contact( #S120.AxisSts.AlarmPresence )
      I_Contact( #Fan_M.MotorSts.AlarmPresence )
      I_Contact( #CIn.ExternalAlarms )
      Not()
      Coil( #Sts.AlarmPresence )
   END_RUNG
   // the same network as SCL:
   #Sts.AlarmPresence := NOT (NOT #Alarm.BrakeTimeOut AND NOT #Alarm.S120_ComErr AND NOT #Alarm.Ax_NotHomed AND NOT #Ax.AxisSts.AlarmPresence AND NOT #S120.AxisSts.AlarmPresence AND NOT #Fan_M.MotorSts.AlarmPresence AND NOT #CIn.ExternalAlarms);
END_REGION

REGION Network 51: Stop aborting
   RUNG wire#powerrail
      Contact( #AreaInterface.Cycle )
      wire#w1
      Contact( #Sts.Standstill )
      wire#w2
      Contact( #Sts.AlarmPresence )
      Coil( #Ctrl.StopAborting )
   END_RUNG
   RUNG wire#w1
      Contact( #Ctrl.StopAborting )
   END_RUNG wire#w2
   RUNG wire#powerrail
      Contact( #AreaInterface.Aut )
   END_RUNG wire#w2
   RUNG wire#powerrail
      Contact( #CIn.Manager.Control_ON )
   END_RUNG wire#w2
   // the same network as SCL:
   #Ctrl.StopAborting := ((#AreaInterface.Cycle AND (#Sts.Standstill OR #Ctrl.StopAborting)) OR #AreaInterface.Aut OR #CIn.Manager.Control_ON) AND #Sts.AlarmPresence;
END_REGION

REGION Network 52 (SCL): Collect machine to zone interface
   #MachineInterface.AutReady := #AreaInterface.Aut AND NOT #Sts.AlarmPresence;
   #MachineInterface.Aborting := #Ctrl.StopAborting;
   #MachineInterface.MotionsStandStill := #TON_NoPendingCmd.Q AND #Sts.Standstill;
   #MachineInterface.AckStopInPhase := #Ctrl.StopInPhase AND #MachineInterface.MotionsStandStill;
   #MachineInterface.AckStopProgrammed := #Ctrl.StopProgrammed AND #MachineInterface.MotionsStandStill;
   #MachineInterface.AlarmsPresence := #Sts.AlarmPresence;
   #MachineInterface.WarningPresence := #Sts.WarningPresence;
END_REGION

REGION Network 53: Warning Machine not ready for automatic
   RUNG wire#powerrail
      Contact( #AreaInterface.CheckAutReady )
      I_Contact( #MachineInterface.AutReady )
      S_SR(operand := #Warning.NotAutReady, r1 := wire#w1)
   END_RUNG
   RUNG wire#powerrail
      Contact( #AreaInterface.Cycle )
   END_RUNG wire#w1
   // the same network as SCL:
   IF #AreaInterface.CheckAutReady AND NOT #MachineInterface.AutReady THEN
       #Warning.NotAutReady := TRUE;   // SR flip-flop
   END_IF;
   IF #AreaInterface.Cycle THEN #Warning.NotAutReady := FALSE; END_IF;
END_REGION

REGION Network 54: +
END_REGION

REGION Network 55: +
END_REGION

REGION Network 56 (SCL): HMI Status Positioning DOL Machine
   // Area dati Status per HMI sull'azionamento

   #HMI.Sts.Enabled :=#S120.AxisSts.Enabled ;
   #HMI.Sts.Standstill := #Sts.Standstill;
   #HMI.Sts.Homed := #COut.Homed;
   #HMI.Sts.Alarm := #Sts.AlarmPresence;
   #HMI.Sts.Warning := #Sts.WarningPresence;
   #HMI.Sts.Plus_Run := #COut.PlusRunning;
   #HMI.Sts.Minus_Run := #COut.MinusRunning;
   #HMI.Sts.InTargetPos := #Ax.AxisSts.InPosition;
   #HMI.Sts.MinPosReached := #COut.MinusLsSwReached OR #COut.MinusLimitReached;
   #HMI.Sts.MaxPosReached := #COut.PlusLsSwReached OR #COut.PlusLimitReached;
   #HMI.Sts.TargetPos := #COut.ActualTargetPos;
   #HMI.Sts.ActualPos := #COut.ActualPosition;
   #HMI.Sts.ActualPos_UM2 := #COut.ActualPosition_UM2;
   #HMI.Sts.ActualVel := #COut.ActualSpeed;
END_REGION

REGION Network 57: +
END_REGION

REGION Network 58: +
END_REGION
END_FUNCTION_BLOCK
